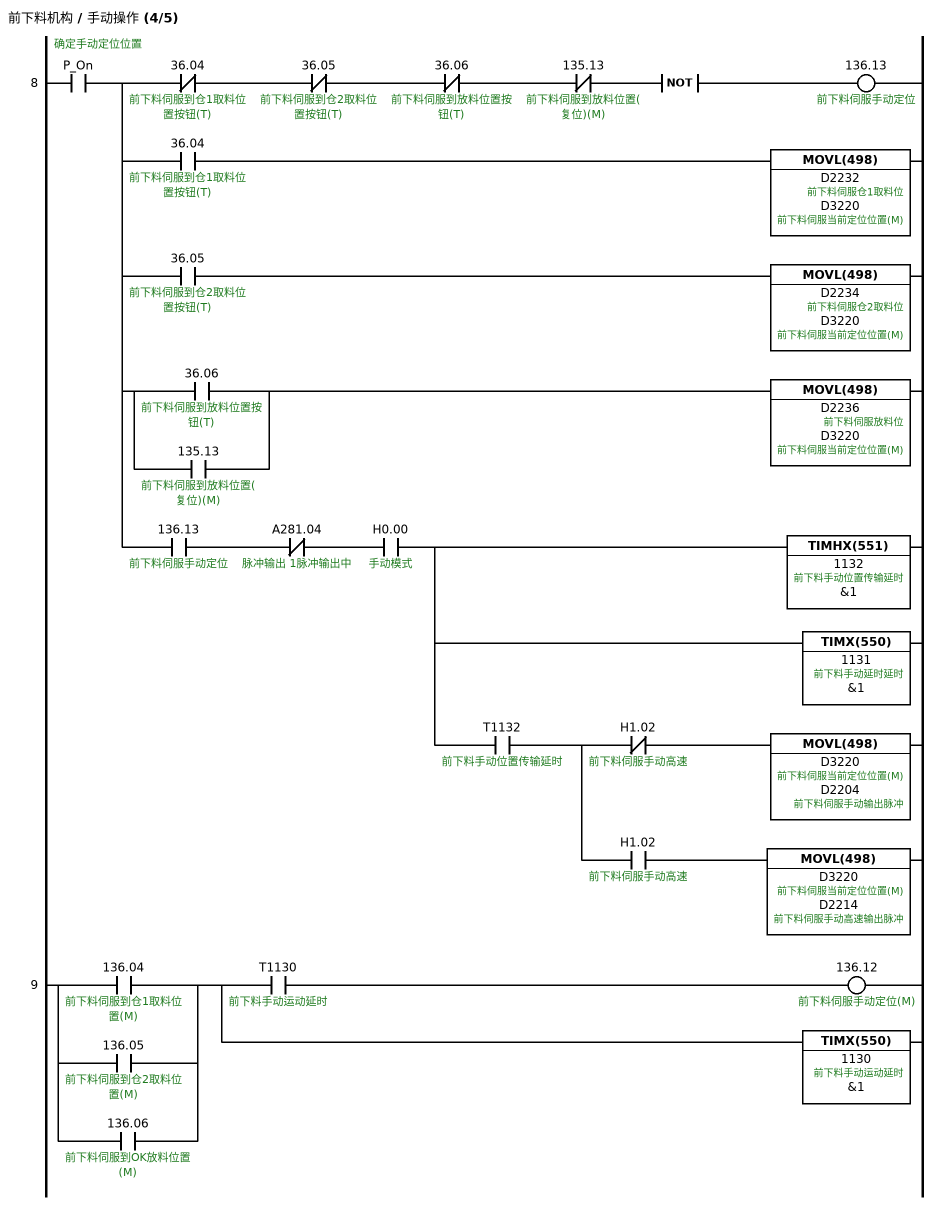
; [picture p168: 前下料机构 / 手动操作, rungs 8-9]
; rung 8: 确定手动定位位置
LD P_On
OUT TR0
ANDNOT 36.04  ; 前下料伺服到仓1取料位置按钮(T)
ANDNOT 36.05  ; 前下料伺服到仓2取料位置按钮(T)
ANDNOT 36.06  ; 前下料伺服到放料位置按钮(T)
ANDNOT 135.13  ; 前下料伺服到放料位置(复位)(M)
NOT(520)
OUT 136.13  ; 前下料伺服手动定位
LD TR0
AND 36.04  ; 前下料伺服到仓1取料位置按钮(T)
MOVL(498) D2232 D3220  ; 前下料伺服仓1取料位, 前下料伺服当前定位位置(M)
LD TR0
AND 36.05  ; 前下料伺服到仓2取料位置按钮(T)
MOVL(498) D2234 D3220  ; 前下料伺服仓2取料位, 前下料伺服当前定位位置(M)
LD TR0
LD 36.06  ; 前下料伺服到放料位置按钮(T)
OR 135.13  ; 前下料伺服到放料位置(复位)(M)
ANDLD
MOVL(498) D2236 D3220  ; 前下料伺服放料位, 前下料伺服当前定位位置(M)
LD TR0
AND 136.13  ; 前下料伺服手动定位
ANDNOT A281.04  ; 脉冲输出 1脉冲输出中
AND H0.00  ; 手动模式
TIMHX(551) 1132 &1  ; 前下料手动位置传输延时
TIMX(550) 1131 &1  ; 前下料手动延时延时
AND T1132  ; 前下料手动位置传输延时
OUT TR0
ANDNOT H1.02  ; 前下料伺服手动高速
MOVL(498) D3220 D2204  ; 前下料伺服当前定位位置(M), 前下料伺服手动输出脉冲
LD TR0
AND H1.02  ; 前下料伺服手动高速
MOVL(498) D3220 D2214  ; 前下料伺服当前定位位置(M), 前下料伺服手动高速输出脉冲
; rung 9
LD 136.04  ; 前下料伺服到仓1取料位置(M)
OR 136.05  ; 前下料伺服到仓2取料位置(M)
OR 136.06  ; 前下料伺服到OK放料位置(M)
OUT TR0
AND T1130  ; 前下料手动运动延时
OUT 136.12  ; 前下料伺服手动定位(M)
LD TR0
TIMX(550) 1130 &1  ; 前下料手动运动延时

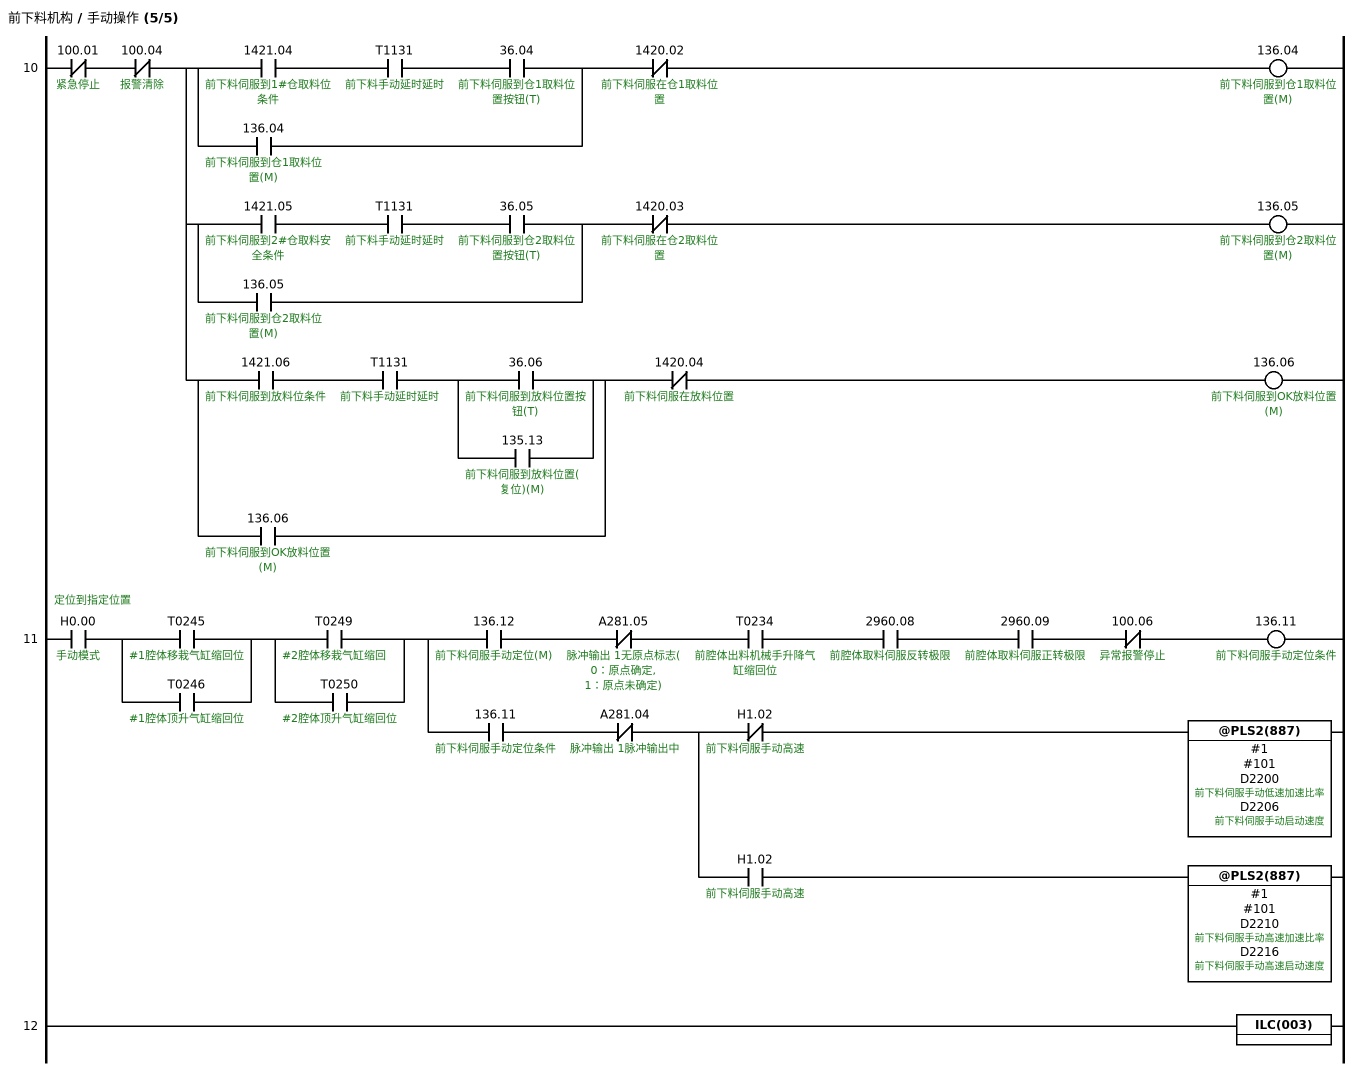
; rung 10
LDNOT 100.01  ; 紧急停止
ANDNOT 100.04  ; 报警清除
OUT TR0
LD 1421.04  ; 前下料伺服到1#仓取料位条件
AND T1131  ; 前下料手动延时延时
AND 36.04  ; 前下料伺服到仓1取料位置按钮(T)
OR 136.04  ; 前下料伺服到仓1取料位置(M)
ANDLD
ANDNOT 1420.02  ; 前下料伺服在仓1取料位置
OUT 136.04  ; 前下料伺服到仓1取料位置(M)
LD TR0
LD 1421.05  ; 前下料伺服到2#仓取料安全条件
AND T1131  ; 前下料手动延时延时
AND 36.05  ; 前下料伺服到仓2取料位置按钮(T)
OR 136.05  ; 前下料伺服到仓2取料位置(M)
ANDLD
ANDNOT 1420.03  ; 前下料伺服在仓2取料位置
OUT 136.05  ; 前下料伺服到仓2取料位置(M)
LD TR0
LD 1421.06  ; 前下料伺服到放料位条件
AND T1131  ; 前下料手动延时延时
LD 36.06  ; 前下料伺服到放料位置按钮(T)
OR 135.13  ; 前下料伺服到放料位置(复位)(M)
ANDLD
OR 136.06  ; 前下料伺服到OK放料位置(M)
ANDLD
ANDNOT 1420.04  ; 前下料伺服在放料位置
OUT 136.06  ; 前下料伺服到OK放料位置(M)
; rung 11: 定位到指定位置
LD H0.00  ; 手动模式
LD T0245  ; #1腔体移栽气缸缩回位
OR T0246  ; #1腔体顶升气缸缩回位
ANDLD
LD T0249  ; #2腔体移栽气缸缩回
OR T0250  ; #2腔体顶升气缸缩回位
ANDLD
OUT TR0
AND 136.12  ; 前下料伺服手动定位(M)
ANDNOT A281.05  ; 脉冲输出 1无原点标志(0：原点确定,1：原点未确定)
AND T0234  ; 前腔体出料机械手升降气缸缩回位
AND 2960.08  ; 前腔体取料伺服反转极限
AND 2960.09  ; 前腔体取料伺服正转极限
ANDNOT 100.06  ; 异常报警停止
OUT 136.11  ; 前下料伺服手动定位条件
LD TR0
AND 136.11  ; 前下料伺服手动定位条件
ANDNOT A281.04  ; 脉冲输出 1脉冲输出中
OUT TR0
ANDNOT H1.02  ; 前下料伺服手动高速
@PLS2(887) #1 #101 D2200 D2206  ; 前下料伺服手动低速加速比率, 前下料伺服手动启动速度
LD TR0
AND H1.02  ; 前下料伺服手动高速
@PLS2(887) #1 #101 D2210 D2216  ; 前下料伺服手动高速加速比率, 前下料伺服手动高速启动速度
; rung 12
ILC(003)

### Section 自动运行

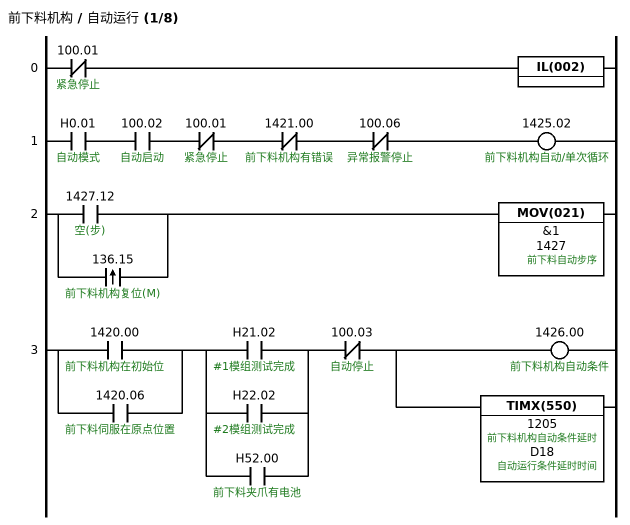
; rung 0
LDNOT 100.01  ; 紧急停止
IL(002)
; rung 1
LD H0.01  ; 自动模式
AND 100.02  ; 自动启动
ANDNOT 100.01  ; 紧急停止
ANDNOT 1421.00  ; 前下料机构有错误
ANDNOT 100.06  ; 异常报警停止
OUT 1425.02  ; 前下料机构自动/单次循环
; rung 2
LD 1427.12  ; 空(步)
@OR 136.15  ; 前下料机构复位(M)
MOV(021) &1 1427  ; 前下料自动步序
; rung 3
LD 1420.00  ; 前下料机构在初始位
OR 1420.06  ; 前下料伺服在原点位置
LD H21.02  ; #1模组测试完成
OR H22.02  ; #2模组测试完成
OR H52.00  ; 前下料夹爪有电池
ANDLD
ANDNOT 100.03  ; 自动停止
OUT 1426.00  ; 前下料机构自动条件
TIMX(550) 1205 D18  ; 自动运行条件延时时间, 前下料机构自动条件延时

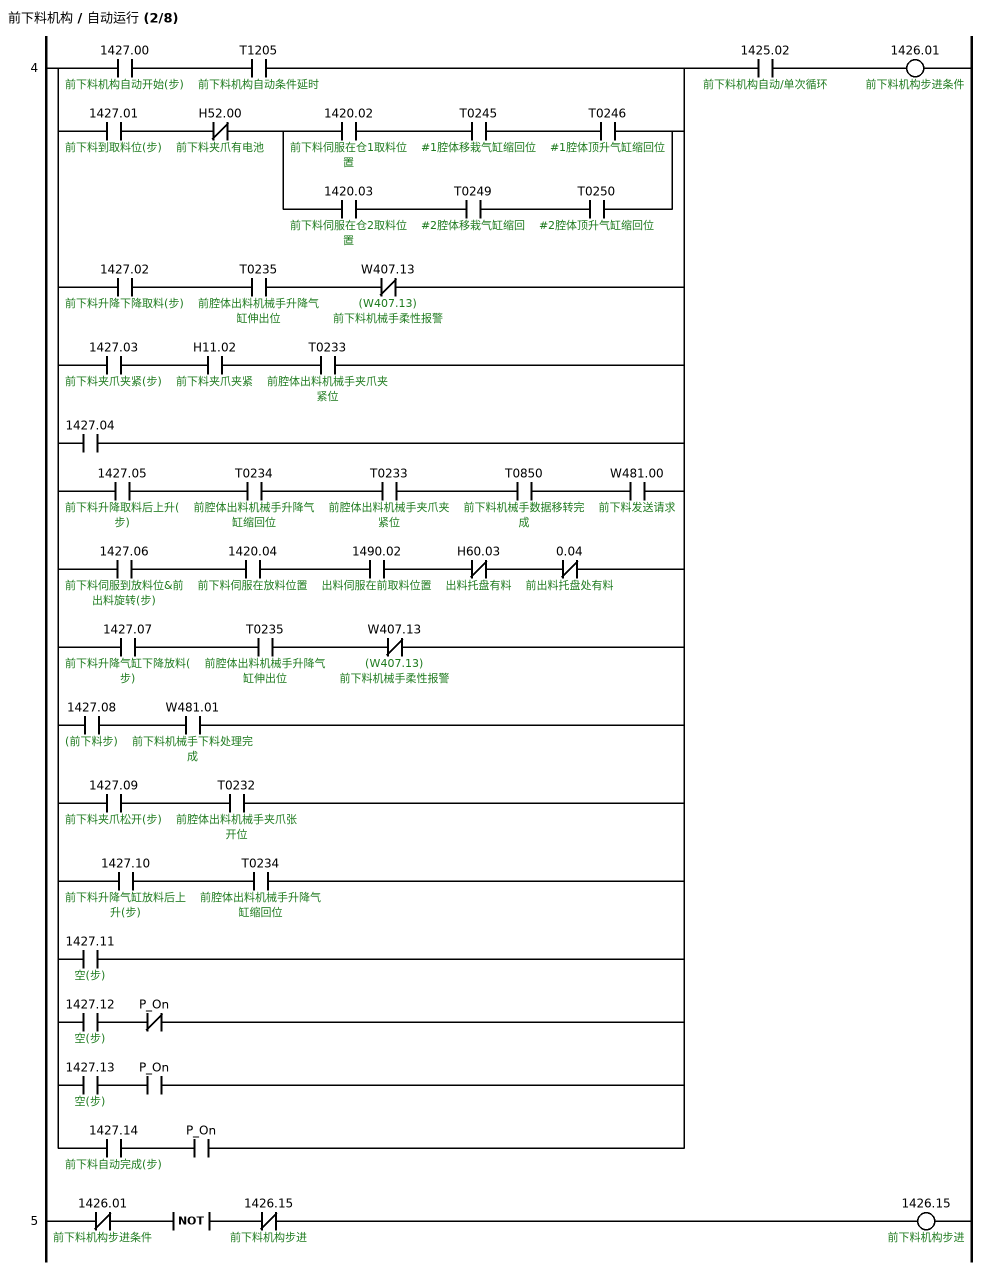
; rung 4
LD 1427.00  ; 前下料机构自动开始(步)
AND T1205  ; 前下料机构自动条件延时
LD 1427.01  ; 前下料到取料位(步)
ANDNOT H52.00  ; 前下料夹爪有电池
LD 1420.02  ; 前下料伺服在仓1取料位置
AND T0245  ; #1腔体移栽气缸缩回位
AND T0246  ; #1腔体顶升气缸缩回位
LD 1420.03  ; 前下料伺服在仓2取料位置
AND T0249  ; #2腔体移栽气缸缩回
AND T0250  ; #2腔体顶升气缸缩回位
ORLD
ANDLD
ORLD
LD 1427.02  ; 前下料升降下降取料(步)
AND T0235  ; 前腔体出料机械手升降气缸伸出位
ANDNOT W407.13  ; (W407.13) 前下料机械手柔性报警
ORLD
LD 1427.03  ; 前下料夹爪夹紧(步)
AND H11.02  ; 前下料夹爪夹紧
AND T0233  ; 前腔体出料机械手夹爪夹紧位
ORLD
OR 1427.04
LD 1427.05  ; 前下料升降取料后上升(步)
AND T0234  ; 前腔体出料机械手升降气缸缩回位
AND T0233  ; 前腔体出料机械手夹爪夹紧位
AND T0850  ; 前下料机械手数据移转完成
AND W481.00  ; 前下料发送请求
ORLD
LD 1427.06  ; 前下料伺服到放料位&前出料旋转(步)
AND 1420.04  ; 前下料伺服在放料位置
AND 1490.02  ; 出料伺服在前取料位置
ANDNOT H60.03  ; 出料托盘有料
ANDNOT 0.04  ; 前出料托盘处有料
ORLD
LD 1427.07  ; 前下料升降气缸下降放料(步)
AND T0235  ; 前腔体出料机械手升降气缸伸出位
ANDNOT W407.13  ; (W407.13) 前下料机械手柔性报警
ORLD
LD 1427.08  ; (前下料步)
AND W481.01  ; 前下料机械手下料处理完成
ORLD
LD 1427.09  ; 前下料夹爪松开(步)
AND T0232  ; 前腔体出料机械手夹爪张开位
ORLD
LD 1427.10  ; 前下料升降气缸放料后上升(步)
AND T0234  ; 前腔体出料机械手升降气缸缩回位
ORLD
OR 1427.11  ; 空(步)
LD 1427.12  ; 空(步)
ANDNOT P_On
ORLD
LD 1427.13  ; 空(步)
AND P_On
ORLD
LD 1427.14  ; 前下料自动完成(步)
AND P_On
ORLD
AND 1425.02  ; 前下料机构自动/单次循环
OUT 1426.01  ; 前下料机构步进条件
; rung 5
LDNOT 1426.01  ; 前下料机构步进条件
NOT(520)
ANDNOT 1426.15  ; 前下料机构步进
OUT 1426.15  ; 前下料机构步进

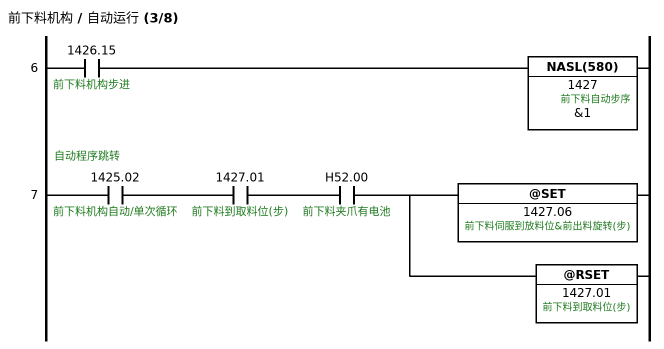
; rung 6
LD 1426.15  ; 前下料机构步进
NASL(580) 1427 &1  ; 前下料自动步序
; rung 7: 自动程序跳转
LD 1425.02  ; 前下料机构自动/单次循环
AND 1427.01  ; 前下料到取料位(步)
AND H52.00  ; 前下料夹爪有电池
@SET 1427.06  ; 前下料伺服到放料位&前出料旋转(步)
@RSET 1427.01  ; 前下料到取料位(步)

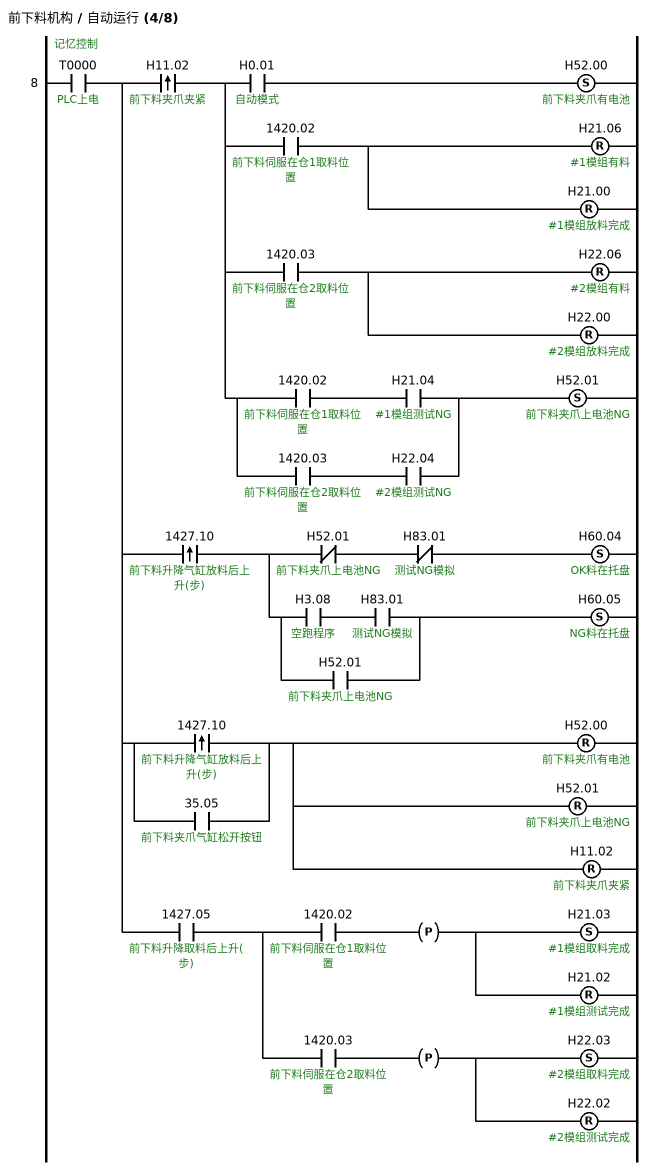
; rung 8: 记忆控制
LD T0000  ; PLC上电
OUT TR0
@AND H11.02  ; 前下料夹爪夹紧
OUT TR1
AND H0.01  ; 自动模式
SET H52.00  ; 前下料夹爪有电池
LD TR1
AND 1420.02  ; 前下料伺服在仓1取料位置
RSET H21.06  ; #1模组有料
RSET H21.00  ; #1模组放料完成
LD TR1
AND 1420.03  ; 前下料伺服在仓2取料位置
RSET H22.06  ; #2模组有料
RSET H22.00  ; #2模组放料完成
LD TR1
LD 1420.02  ; 前下料伺服在仓1取料位置
AND H21.04  ; #1模组测试NG
LD 1420.03  ; 前下料伺服在仓2取料位置
AND H22.04  ; #2模组测试NG
ORLD
ANDLD
SET H52.01  ; 前下料夹爪上电池NG
LD TR0
@AND 1427.10  ; 前下料升降气缸放料后上升(步)
OUT TR1
ANDNOT H52.01  ; 前下料夹爪上电池NG
ANDNOT H83.01  ; 测试NG模拟
SET H60.04  ; OK料在托盘
LD TR1
LD H3.08  ; 空跑程序
AND H83.01  ; 测试NG模拟
OR H52.01  ; 前下料夹爪上电池NG
ANDLD
SET H60.05  ; NG料在托盘
LD TR0
@LD 1427.10  ; 前下料升降气缸放料后上升(步)
OR 35.05  ; 前下料夹爪气缸松开按钮
ANDLD
RSET H52.00  ; 前下料夹爪有电池
RSET H52.01  ; 前下料夹爪上电池NG
RSET H11.02  ; 前下料夹爪夹紧
LD TR0
AND 1427.05  ; 前下料升降取料后上升(步)
OUT TR0
AND 1420.02  ; 前下料伺服在仓1取料位置
UP(521)
SET H21.03  ; #1模组取料完成
RSET H21.02  ; #1模组测试完成
LD TR0
AND 1420.03  ; 前下料伺服在仓2取料位置
UP(521)
SET H22.03  ; #2模组取料完成
RSET H22.02  ; #2模组测试完成

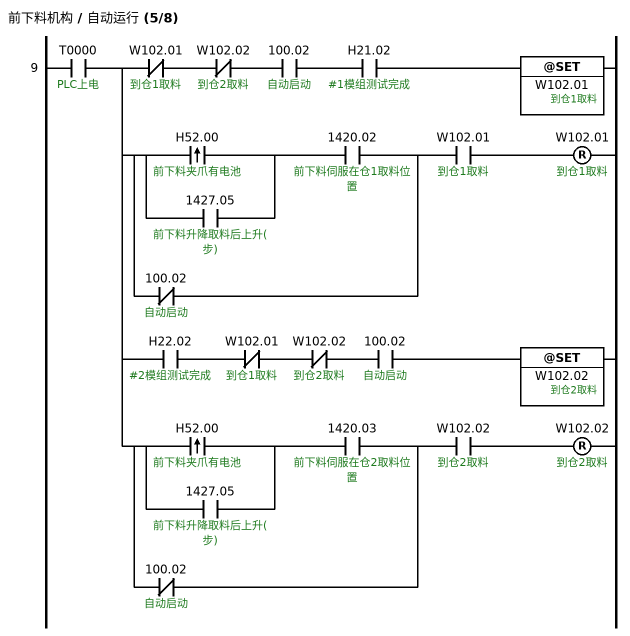
; rung 9
LD T0000  ; PLC上电
OUT TR0
ANDNOT W102.01  ; 到仓1取料
ANDNOT W102.02  ; 到仓2取料
AND 100.02  ; 自动启动
AND H21.02  ; #1模组测试完成
@SET W102.01  ; 到仓1取料
LD TR0
@LD H52.00  ; 前下料夹爪有电池
OR 1427.05  ; 前下料升降取料后上升(步)
AND 1420.02  ; 前下料伺服在仓1取料位置
ORNOT 100.02  ; 自动启动
ANDLD
AND W102.01  ; 到仓1取料
RSET W102.01  ; 到仓1取料
LD TR0
AND H22.02  ; #2模组测试完成
ANDNOT W102.01  ; 到仓1取料
ANDNOT W102.02  ; 到仓2取料
AND 100.02  ; 自动启动
@SET W102.02  ; 到仓2取料
LD TR0
@LD H52.00  ; 前下料夹爪有电池
OR 1427.05  ; 前下料升降取料后上升(步)
AND 1420.03  ; 前下料伺服在仓2取料位置
ORNOT 100.02  ; 自动启动
ANDLD
AND W102.02  ; 到仓2取料
RSET W102.02  ; 到仓2取料

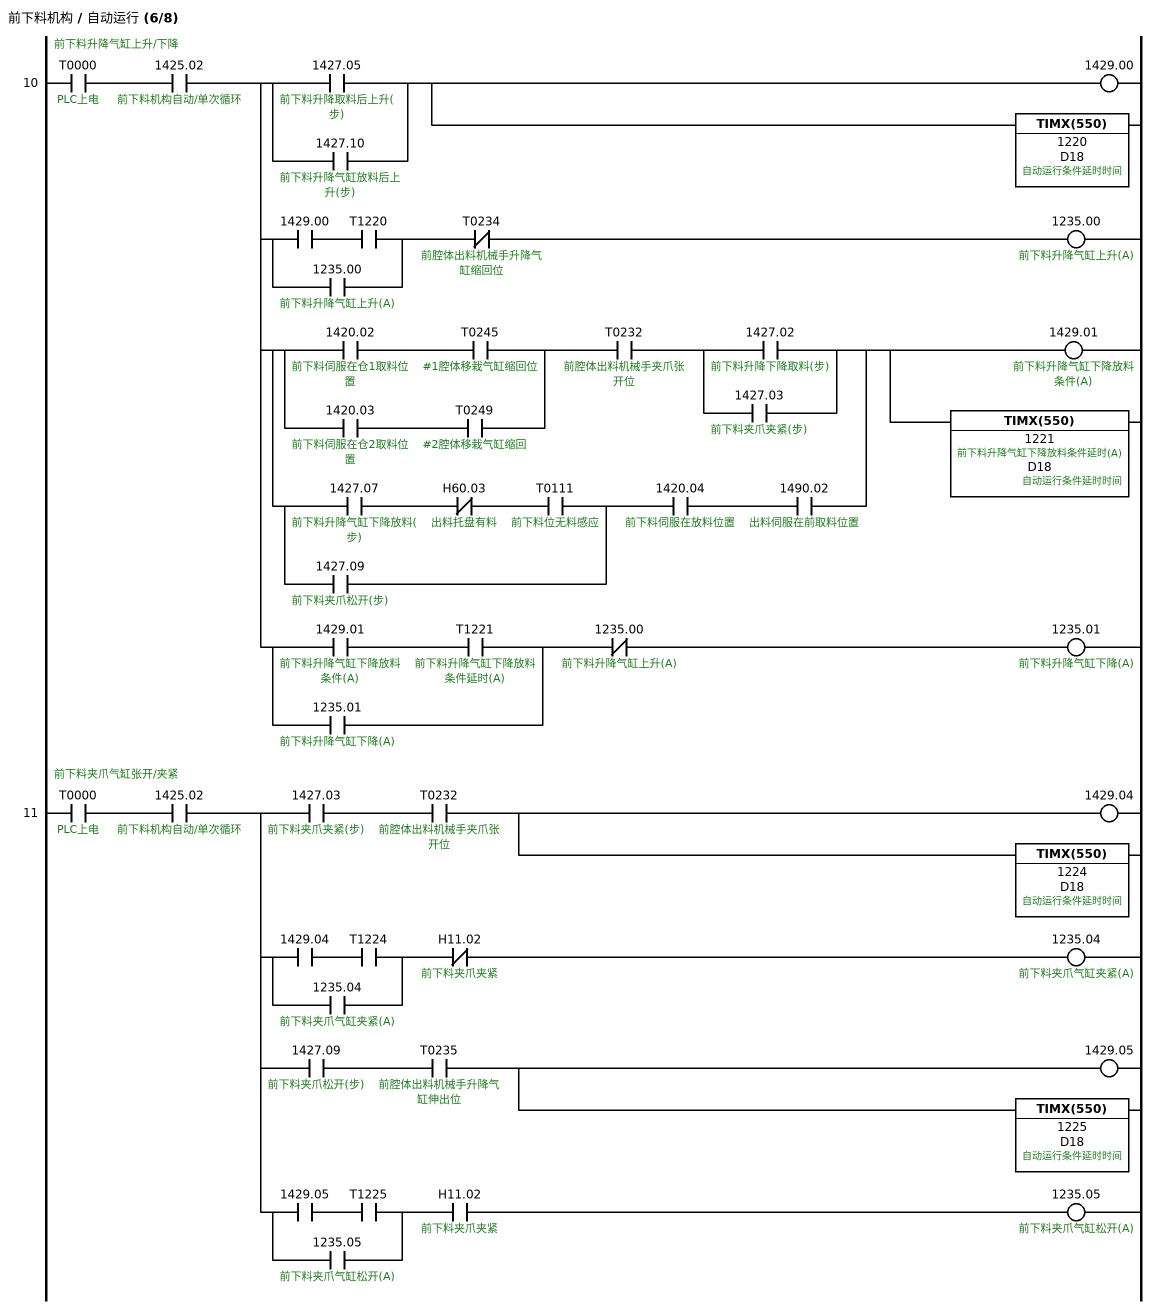
; rung 10: 前下料升降气缸上升/下降
LD T0000  ; PLC上电
AND 1425.02  ; 前下料机构自动/单次循环
OUT TR0
LD 1427.05  ; 前下料升降取料后上升(步)
OR 1427.10  ; 前下料升降气缸放料后上升(步)
ANDLD
OUT 1429.00
TIMX(550) 1220 D18  ; 自动运行条件延时时间
LD TR0
LD 1429.00
AND T1220
OR 1235.00  ; 前下料升降气缸上升(A)
ANDLD
ANDNOT T0234  ; 前腔体出料机械手升降气缸缩回位
OUT 1235.00  ; 前下料升降气缸上升(A)
LD TR0
LD 1420.02  ; 前下料伺服在仓1取料位置
AND T0245  ; #1腔体移栽气缸缩回位
LD 1420.03  ; 前下料伺服在仓2取料位置
AND T0249  ; #2腔体移栽气缸缩回
ORLD
AND T0232  ; 前腔体出料机械手夹爪张开位
LD 1427.02  ; 前下料升降下降取料(步)
OR 1427.03  ; 前下料夹爪夹紧(步)
ANDLD
LD 1427.07  ; 前下料升降气缸下降放料(步)
ANDNOT H60.03  ; 出料托盘有料
AND T0111  ; 前下料位无料感应
OR 1427.09  ; 前下料夹爪松开(步)
AND 1420.04  ; 前下料伺服在放料位置
AND 1490.02  ; 出料伺服在前取料位置
ORLD
ANDLD
OUT 1429.01  ; 前下料升降气缸下降放料条件(A)
TIMX(550) 1221 D18  ; 自动运行条件延时时间, 前下料升降气缸下降放料条件延时(A)
LD TR0
LD 1429.01  ; 前下料升降气缸下降放料条件(A)
AND T1221  ; 前下料升降气缸下降放料条件延时(A)
OR 1235.01  ; 前下料升降气缸下降(A)
ANDLD
ANDNOT 1235.00  ; 前下料升降气缸上升(A)
OUT 1235.01  ; 前下料升降气缸下降(A)
; rung 11: 前下料夹爪气缸张开/夹紧
LD T0000  ; PLC上电
AND 1425.02  ; 前下料机构自动/单次循环
OUT TR0
AND 1427.03  ; 前下料夹爪夹紧(步)
AND T0232  ; 前腔体出料机械手夹爪张开位
OUT 1429.04
TIMX(550) 1224 D18  ; 自动运行条件延时时间
LD TR0
LD 1429.04
AND T1224
OR 1235.04  ; 前下料夹爪气缸夹紧(A)
ANDLD
ANDNOT H11.02  ; 前下料夹爪夹紧
OUT 1235.04  ; 前下料夹爪气缸夹紧(A)
LD TR0
AND 1427.09  ; 前下料夹爪松开(步)
AND T0235  ; 前腔体出料机械手升降气缸伸出位
OUT 1429.05
TIMX(550) 1225 D18  ; 自动运行条件延时时间
LD TR0
LD 1429.05
AND T1225
OR 1235.05  ; 前下料夹爪气缸松开(A)
ANDLD
AND H11.02  ; 前下料夹爪夹紧
OUT 1235.05  ; 前下料夹爪气缸松开(A)

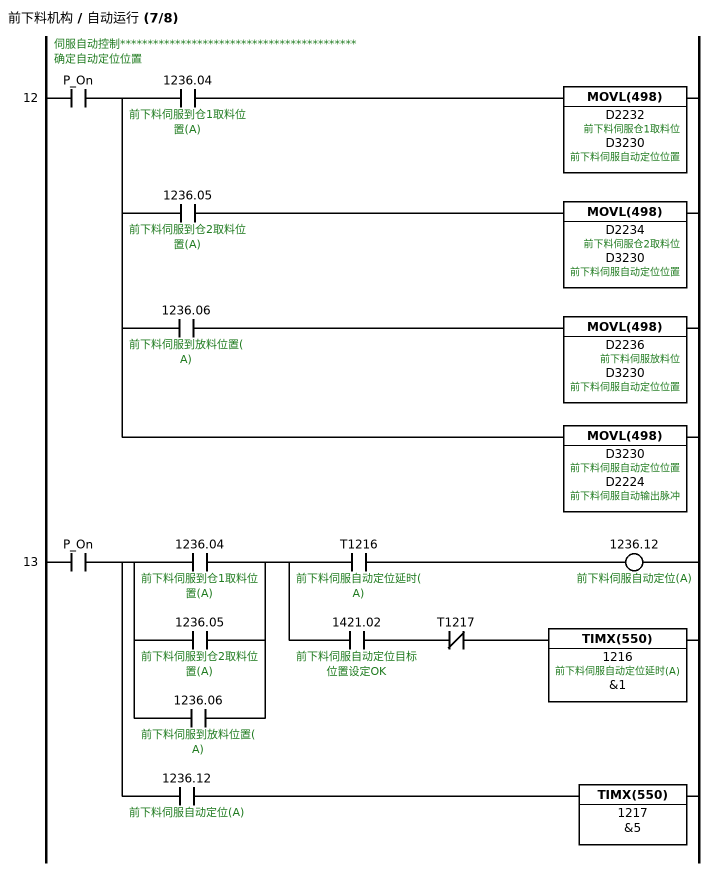
; rung 12: 伺服自动控制******************************************* / 确定自动定位位置
LD P_On
OUT TR0
AND 1236.04  ; 前下料伺服到仓1取料位置(A)
MOVL(498) D2232 D3230  ; 前下料伺服仓1取料位, 前下料伺服自动定位位置
LD TR0
AND 1236.05  ; 前下料伺服到仓2取料位置(A)
MOVL(498) D2234 D3230  ; 前下料伺服仓2取料位, 前下料伺服自动定位位置
LD TR0
AND 1236.06  ; 前下料伺服到放料位置(A)
MOVL(498) D2236 D3230  ; 前下料伺服放料位, 前下料伺服自动定位位置
LD TR0
MOVL(498) D3230 D2224  ; 前下料伺服自动定位位置, 前下料伺服自动输出脉冲
; rung 13
LD P_On
OUT TR0
LD 1236.04  ; 前下料伺服到仓1取料位置(A)
OR 1236.05  ; 前下料伺服到仓2取料位置(A)
OR 1236.06  ; 前下料伺服到放料位置(A)
ANDLD
OUT TR1
AND T1216  ; 前下料伺服自动定位延时(A)
OUT 1236.12  ; 前下料伺服自动定位(A)
LD TR1
AND 1421.02  ; 前下料伺服自动定位目标位置设定OK
ANDNOT T1217
TIMX(550) 1216 &1  ; 前下料伺服自动定位延时(A)
LD TR0
AND 1236.12  ; 前下料伺服自动定位(A)
TIMX(550) 1217 &5

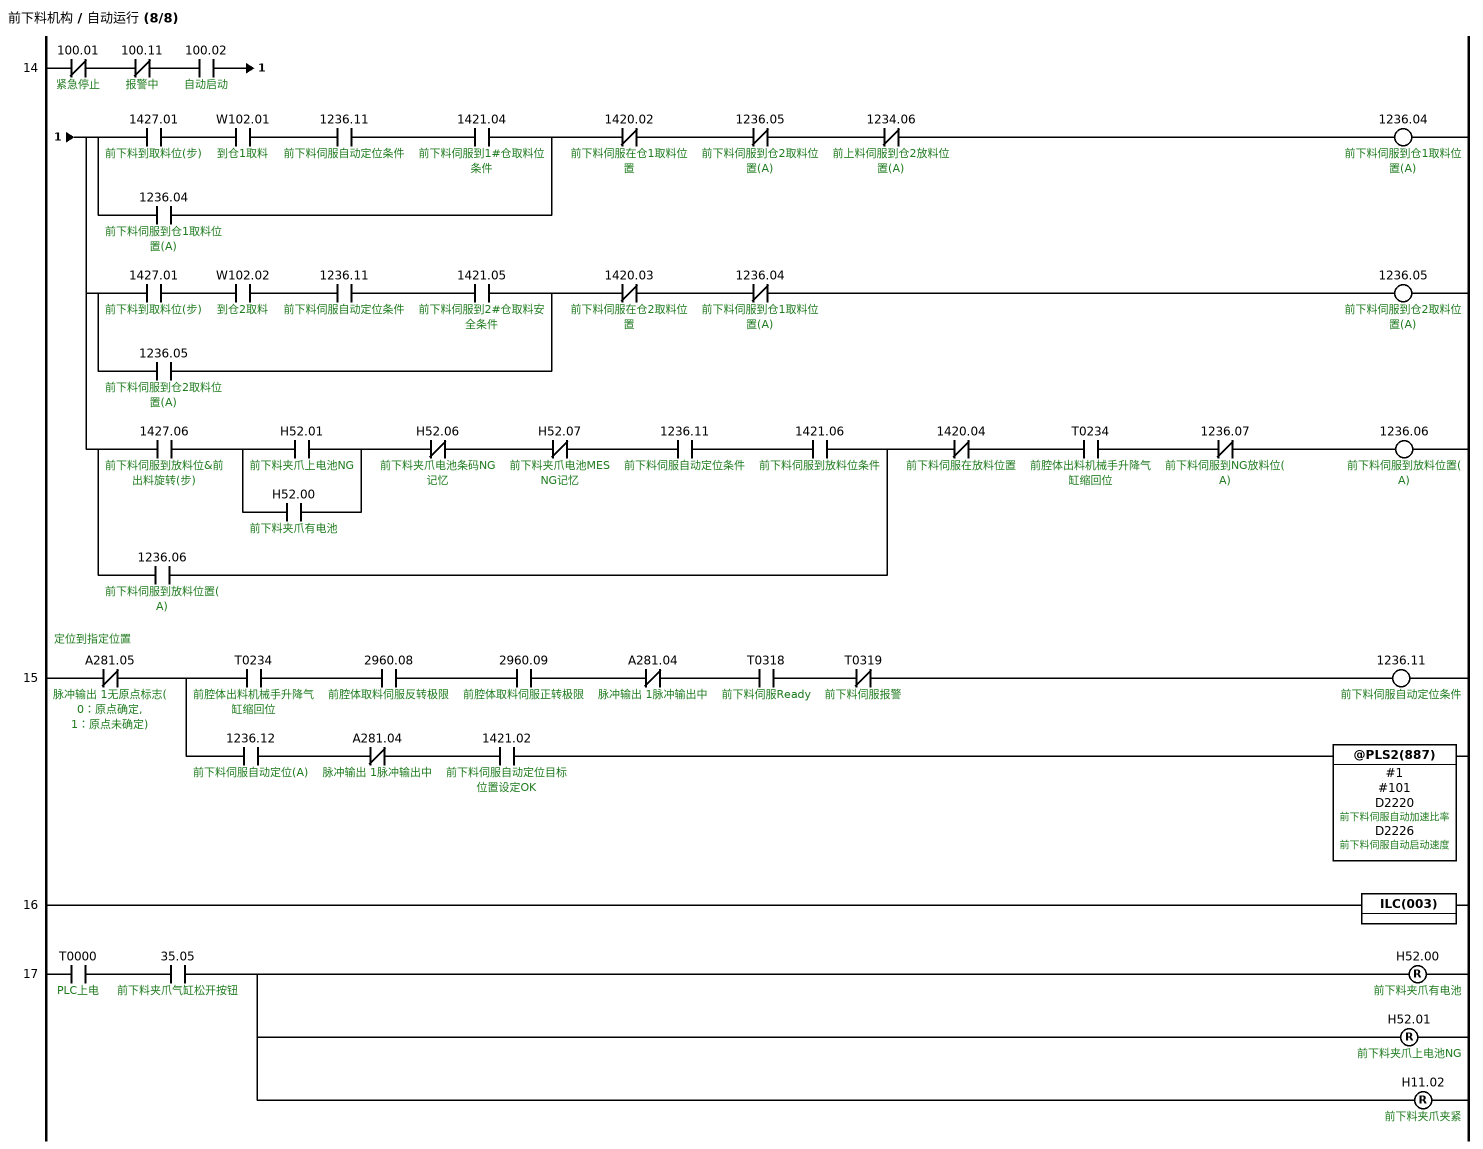
; rung 14
LDNOT 100.01  ; 紧急停止
ANDNOT 100.11  ; 报警中
AND 100.02  ; 自动启动
OUT TR0
LD 1427.01  ; 前下料到取料位(步)
AND W102.01  ; 到仓1取料
AND 1236.11  ; 前下料伺服自动定位条件
AND 1421.04  ; 前下料伺服到1#仓取料位条件
OR 1236.04  ; 前下料伺服到仓1取料位置(A)
ANDLD
ANDNOT 1420.02  ; 前下料伺服在仓1取料位置
ANDNOT 1236.05  ; 前下料伺服到仓2取料位置(A)
ANDNOT 1234.06  ; 前上料伺服到仓2放料位置(A)
OUT 1236.04  ; 前下料伺服到仓1取料位置(A)
LD TR0
LD 1427.01  ; 前下料到取料位(步)
AND W102.02  ; 到仓2取料
AND 1236.11  ; 前下料伺服自动定位条件
AND 1421.05  ; 前下料伺服到2#仓取料安全条件
OR 1236.05  ; 前下料伺服到仓2取料位置(A)
ANDLD
ANDNOT 1420.03  ; 前下料伺服在仓2取料位置
ANDNOT 1236.04  ; 前下料伺服到仓1取料位置(A)
OUT 1236.05  ; 前下料伺服到仓2取料位置(A)
LD TR0
LD 1427.06  ; 前下料伺服到放料位&前出料旋转(步)
LD H52.01  ; 前下料夹爪上电池NG
OR H52.00  ; 前下料夹爪有电池
ANDLD
ANDNOT H52.06  ; 前下料夹爪电池条码NG记忆
ANDNOT H52.07  ; 前下料夹爪电池MES NG记忆
AND 1236.11  ; 前下料伺服自动定位条件
AND 1421.06  ; 前下料伺服到放料位条件
OR 1236.06  ; 前下料伺服到放料位置(A)
ANDLD
ANDNOT 1420.04  ; 前下料伺服在放料位置
AND T0234  ; 前腔体出料机械手升降气缸缩回位
ANDNOT 1236.07  ; 前下料伺服到NG放料位(A)
OUT 1236.06  ; 前下料伺服到放料位置(A)
; rung 15: 定位到指定位置
LDNOT A281.05  ; 脉冲输出 1无原点标志(0：原点确定,1：原点未确定)
OUT TR0
AND T0234  ; 前腔体出料机械手升降气缸缩回位
AND 2960.08  ; 前腔体取料伺服反转极限
AND 2960.09  ; 前腔体取料伺服正转极限
ANDNOT A281.04  ; 脉冲输出 1脉冲输出中
AND T0318  ; 前下料伺服Ready
ANDNOT T0319  ; 前下料伺服报警
OUT 1236.11  ; 前下料伺服自动定位条件
LD TR0
AND 1236.12  ; 前下料伺服自动定位(A)
ANDNOT A281.04  ; 脉冲输出 1脉冲输出中
AND 1421.02  ; 前下料伺服自动定位目标位置设定OK
@PLS2(887) #1 #101 D2220 D2226  ; 前下料伺服自动加速比率, 前下料伺服自动启动速度
; rung 16
ILC(003)
; rung 17
LD T0000  ; PLC上电
AND 35.05  ; 前下料夹爪气缸松开按钮
RSET H52.00  ; 前下料夹爪有电池
RSET H52.01  ; 前下料夹爪上电池NG
RSET H11.02  ; 前下料夹爪夹紧

### Section 外部输出

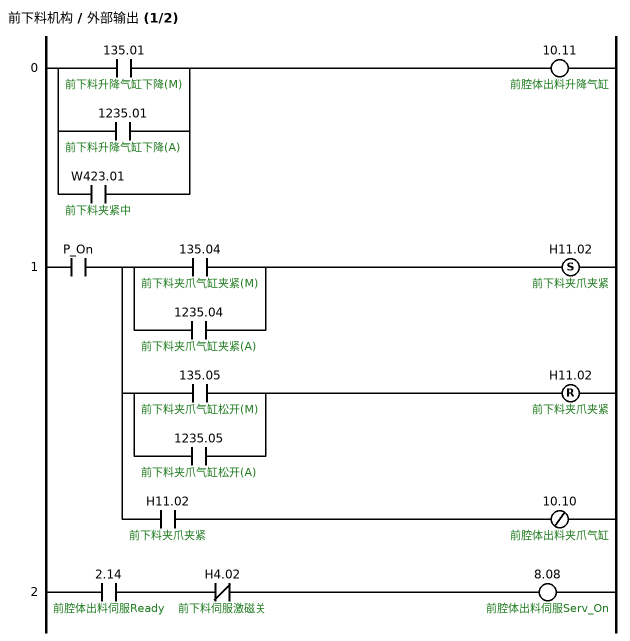
; rung 0
LD 135.01  ; 前下料升降气缸下降(M)
OR 1235.01  ; 前下料升降气缸下降(A)
OR W423.01  ; 前下料夹紧中
OUT 10.11  ; 前腔体出料升降气缸
; rung 1
LD P_On
OUT TR0
LD 135.04  ; 前下料夹爪气缸夹紧(M)
OR 1235.04  ; 前下料夹爪气缸夹紧(A)
ANDLD
SET H11.02  ; 前下料夹爪夹紧
LD TR0
LD 135.05  ; 前下料夹爪气缸松开(M)
OR 1235.05  ; 前下料夹爪气缸松开(A)
ANDLD
RSET H11.02  ; 前下料夹爪夹紧
LD TR0
AND H11.02  ; 前下料夹爪夹紧
OUTNOT 10.10  ; 前腔体出料夹爪气缸
; rung 2
LD 2.14  ; 前腔体出料伺服Ready
ANDNOT H4.02  ; 前下料伺服激磁关
OUT 8.08  ; 前腔体出料伺服Serv_On

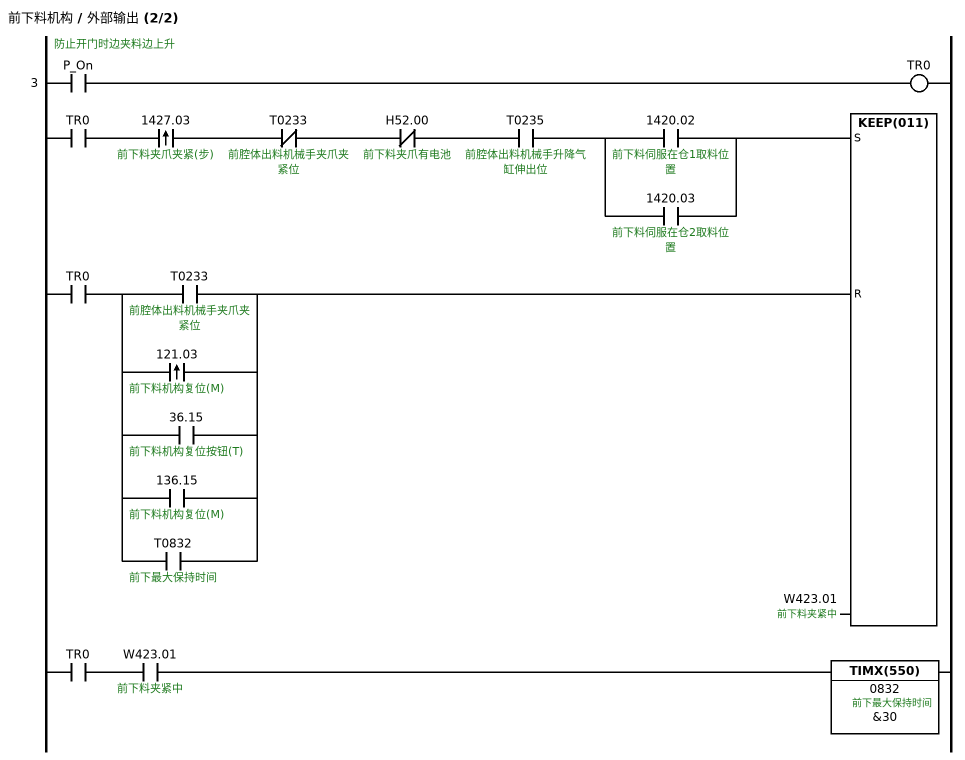
; rung 3: 防止开门时边夹料边上升
LD P_On
OUT TR0
@AND 1427.03  ; 前下料夹爪夹紧(步)
ANDNOT T0233  ; 前腔体出料机械手夹爪夹紧位
ANDNOT H52.00  ; 前下料夹爪有电池
AND T0235  ; 前腔体出料机械手升降气缸伸出位
LD 1420.02  ; 前下料伺服在仓1取料位置
OR 1420.03  ; 前下料伺服在仓2取料位置
ANDLD
LD TR0
LD T0233  ; 前腔体出料机械手夹爪夹紧位
@OR 121.03  ; 前下料机构复位(M)
OR 36.15  ; 前下料机构复位按钮(T)
OR 136.15  ; 前下料机构复位(M)
OR T0832  ; 前下最大保持时间
ANDLD
KEEP(011) W423.01  ; 前下料夹紧中
LD TR0
AND W423.01  ; 前下料夹紧中
TIMX(550) 0832 &30  ; 前下最大保持时间

### Section 进出机构外部输出

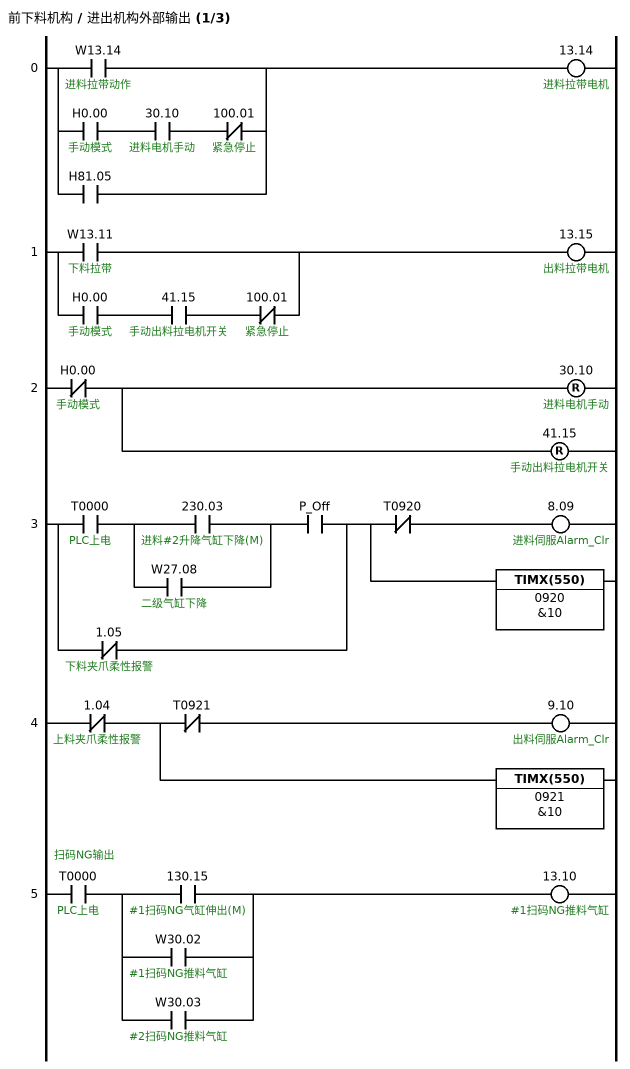
; rung 0
LD W13.14  ; 进料拉带动作
LD H0.00  ; 手动模式
AND 30.10  ; 进料电机手动
ANDNOT 100.01  ; 紧急停止
ORLD
OR H81.05
OUT 13.14  ; 进料拉带电机
; rung 1
LD W13.11  ; 下料拉带
LD H0.00  ; 手动模式
AND 41.15  ; 手动出料拉电机开关
ANDNOT 100.01  ; 紧急停止
ORLD
OUT 13.15  ; 出料拉带电机
; rung 2
LDNOT H0.00  ; 手动模式
RSET 30.10  ; 进料电机手动
RSET 41.15  ; 手动出料拉电机开关
; rung 3
LD T0000  ; PLC上电
LD 230.03  ; 进料#2升降气缸下降(M)
OR W27.08  ; 二级气缸下降
ANDLD
AND P_Off
ORNOT 1.05  ; 下料夹爪柔性报警
OUT TR0
ANDNOT T0920
OUT 8.09  ; 进料伺服Alarm_Clr
LD TR0
TIMX(550) 0920 &10
; rung 4
LDNOT 1.04  ; 上料夹爪柔性报警
OUT TR0
ANDNOT T0921
OUT 9.10  ; 出料伺服Alarm_Clr
LD TR0
TIMX(550) 0921 &10
; rung 5: 扫码NG输出
LD T0000  ; PLC上电
LD 130.15  ; #1扫码NG气缸伸出(M)
OR W30.02  ; #1扫码NG推料气缸
OR W30.03  ; #2扫码NG推料气缸
ANDLD
OUT 13.10  ; #1扫码NG推料气缸

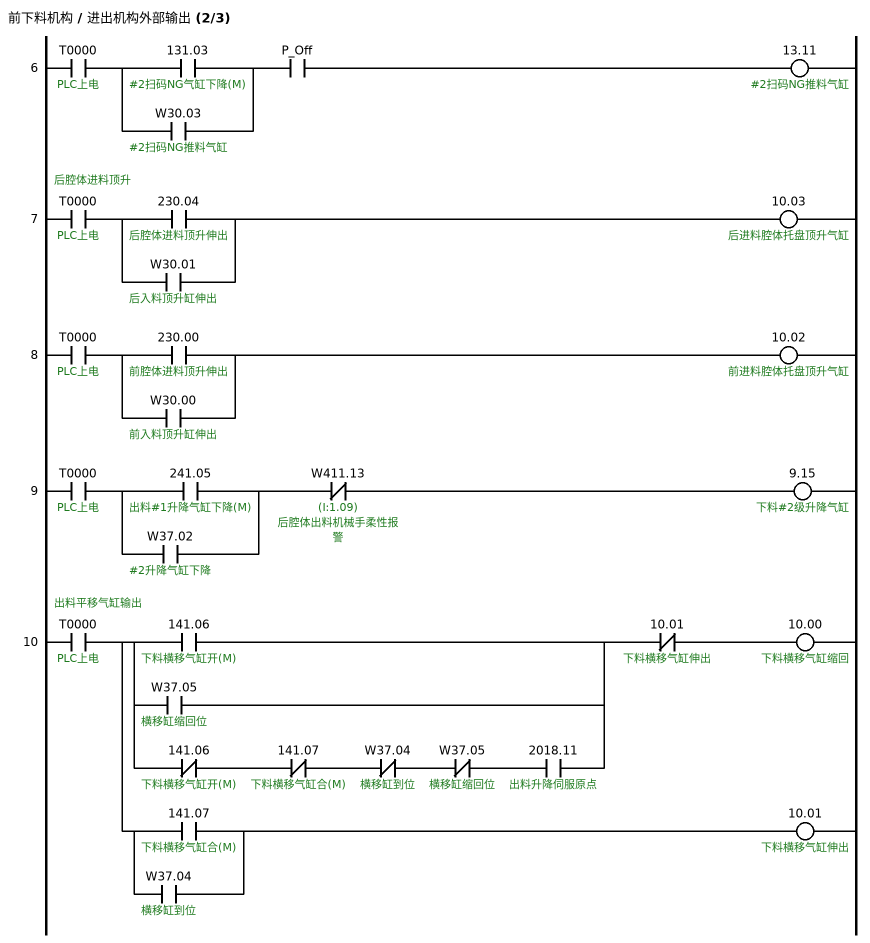
; rung 6
LD T0000  ; PLC上电
LD 131.03  ; #2扫码NG气缸下降(M)
OR W30.03  ; #2扫码NG推料气缸
ANDLD
AND P_Off
OUT 13.11  ; #2扫码NG推料气缸
; rung 7: 后腔体进料顶升
LD T0000  ; PLC上电
LD 230.04  ; 后腔体进料顶升伸出
OR W30.01  ; 后入料顶升缸伸出
ANDLD
OUT 10.03  ; 后进料腔体托盘顶升气缸
; rung 8
LD T0000  ; PLC上电
LD 230.00  ; 前腔体进料顶升伸出
OR W30.00  ; 前入料顶升缸伸出
ANDLD
OUT 10.02  ; 前进料腔体托盘顶升气缸
; rung 9
LD T0000  ; PLC上电
LD 241.05  ; 出料#1升降气缸下降(M)
OR W37.02  ; #2升降气缸下降
ANDLD
ANDNOT W411.13  ; (I:1.09) 后腔体出料机械手柔性报警
OUT 9.15  ; 下料#2级升降气缸
; rung 10: 出料平移气缸输出
LD T0000  ; PLC上电
OUT TR0
LD 141.06  ; 下料横移气缸开(M)
OR W37.05  ; 横移缸缩回位
LDNOT 141.06  ; 下料横移气缸开(M)
ANDNOT 141.07  ; 下料横移气缸合(M)
ANDNOT W37.04  ; 横移缸到位
ANDNOT W37.05  ; 横移缸缩回位
AND 2018.11  ; 出料升降伺服原点
ORLD
ANDLD
ANDNOT 10.01  ; 下料横移气缸伸出
OUT 10.00  ; 下料横移气缸缩回
LD TR0
LD 141.07  ; 下料横移气缸合(M)
OR W37.04  ; 横移缸到位
ANDLD
OUT 10.01  ; 下料横移气缸伸出

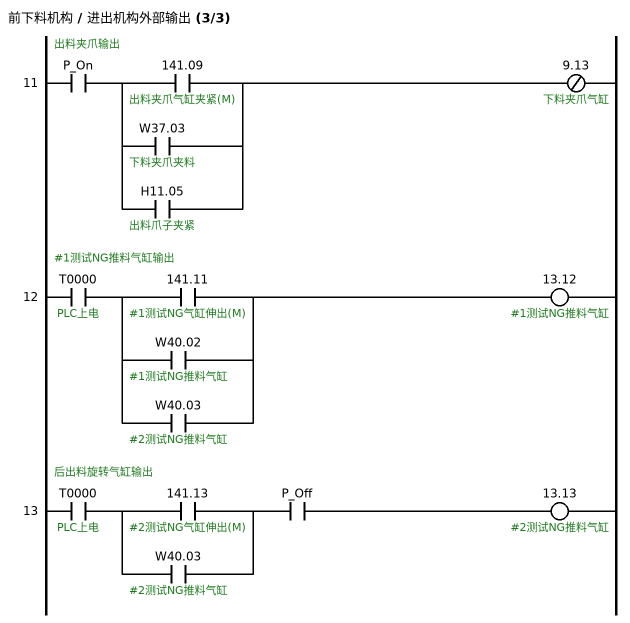
; rung 11: 出料夹爪输出
LD P_On
LD 141.09  ; 出料夹爪气缸夹紧(M)
OR W37.03  ; 下料夹爪夹料
OR H11.05  ; 出料爪子夹紧
ANDLD
OUTNOT 9.13  ; 下料夹爪气缸
; rung 12: #1测试NG推料气缸输出
LD T0000  ; PLC上电
LD 141.11  ; #1测试NG气缸伸出(M)
OR W40.02  ; #1测试NG推料气缸
OR W40.03  ; #2测试NG推料气缸
ANDLD
OUT 13.12  ; #1测试NG推料气缸
; rung 13: 后出料旋转气缸输出
LD T0000  ; PLC上电
LD 141.13  ; #2测试NG气缸伸出(M)
OR W40.03  ; #2测试NG推料气缸
ANDLD
AND P_Off
OUT 13.13  ; #2测试NG推料气缸

### Section 指示灯
; rung 0: ************************************************** / 气缸动作及位置指示灯

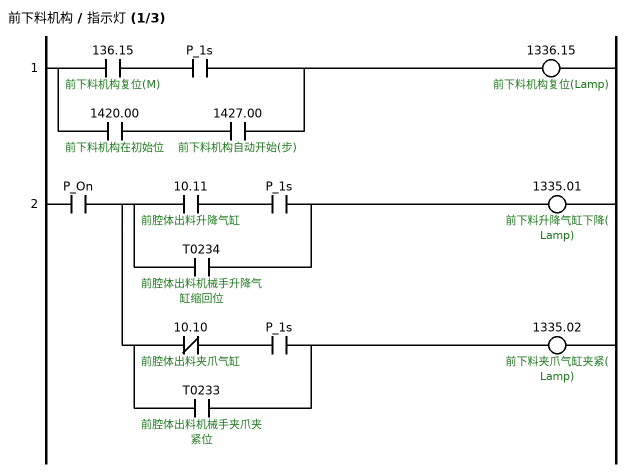
; rung 1
LD 136.15  ; 前下料机构复位(M)
AND P_1s
LD 1420.00  ; 前下料机构在初始位
AND 1427.00  ; 前下料机构自动开始(步)
ORLD
OUT 1336.15  ; 前下料机构复位(Lamp)
; rung 2
LD P_On
OUT TR0
LD 10.11  ; 前腔体出料升降气缸
AND P_1s
OR T0234  ; 前腔体出料机械手升降气缸缩回位
ANDLD
OUT 1335.01  ; 前下料升降气缸下降(Lamp)
LD TR0
LDNOT 10.10  ; 前腔体出料夹爪气缸
AND P_1s
OR T0233  ; 前腔体出料机械手夹爪夹紧位
ANDLD
OUT 1335.02  ; 前下料夹爪气缸夹紧(Lamp)

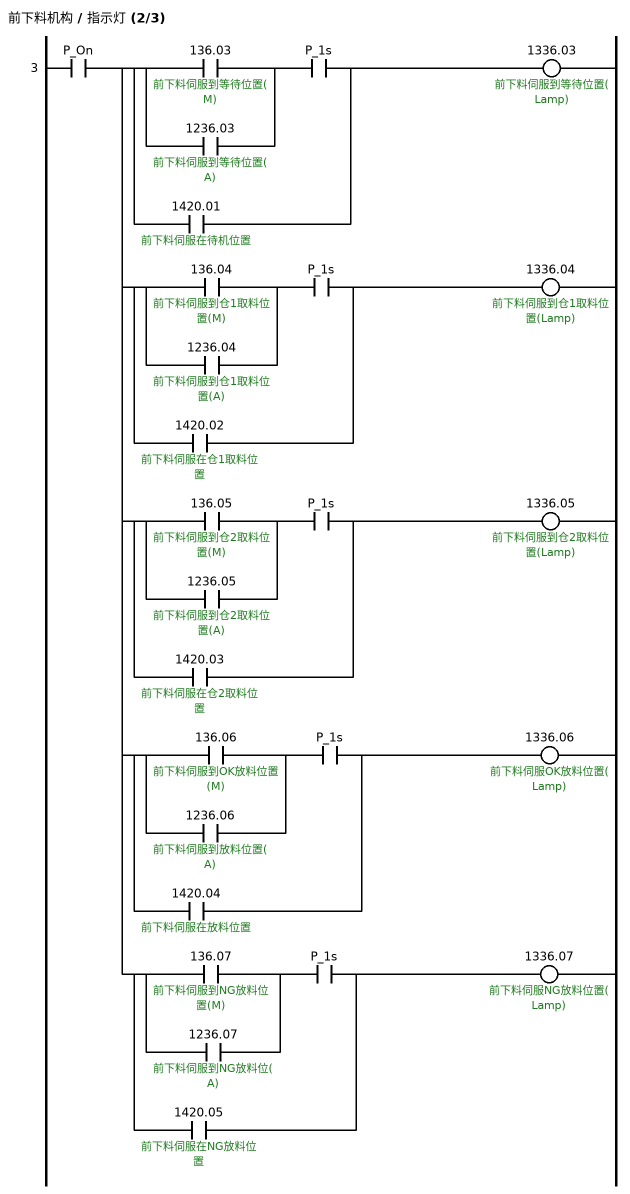
; rung 3
LD P_On
OUT TR0
LD 136.03  ; 前下料伺服到等待位置(M)
OR 1236.03  ; 前下料伺服到等待位置(A)
AND P_1s
OR 1420.01  ; 前下料伺服在待机位置
ANDLD
OUT 1336.03  ; 前下料伺服到等待位置(Lamp)
LD TR0
LD 136.04  ; 前下料伺服到仓1取料位置(M)
OR 1236.04  ; 前下料伺服到仓1取料位置(A)
AND P_1s
OR 1420.02  ; 前下料伺服在仓1取料位置
ANDLD
OUT 1336.04  ; 前下料伺服到仓1取料位置(Lamp)
LD TR0
LD 136.05  ; 前下料伺服到仓2取料位置(M)
OR 1236.05  ; 前下料伺服到仓2取料位置(A)
AND P_1s
OR 1420.03  ; 前下料伺服在仓2取料位置
ANDLD
OUT 1336.05  ; 前下料伺服到仓2取料位置(Lamp)
LD TR0
LD 136.06  ; 前下料伺服到OK放料位置(M)
OR 1236.06  ; 前下料伺服到放料位置(A)
AND P_1s
OR 1420.04  ; 前下料伺服在放料位置
ANDLD
OUT 1336.06  ; 前下料伺服OK放料位置(Lamp)
LD TR0
LD 136.07  ; 前下料伺服到NG放料位置(M)
OR 1236.07  ; 前下料伺服到NG放料位(A)
AND P_1s
OR 1420.05  ; 前下料伺服在NG放料位置
ANDLD
OUT 1336.07  ; 前下料伺服NG放料位置(Lamp)

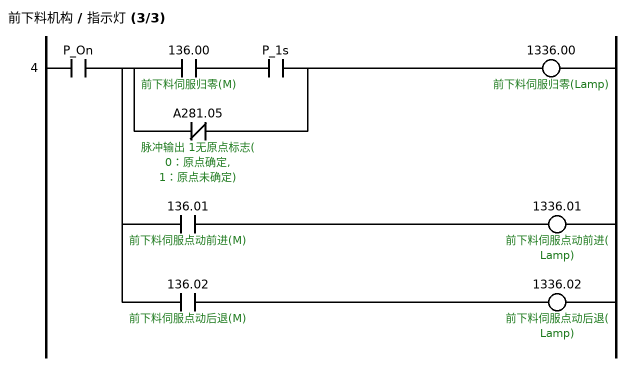
; rung 4
LD P_On
OUT TR0
LD 136.00  ; 前下料伺服归零(M)
AND P_1s
ORNOT A281.05  ; 脉冲输出 1无原点标志(0：原点确定,1：原点未确定)
ANDLD
OUT 1336.00  ; 前下料伺服归零(Lamp)
LD TR0
AND 136.01  ; 前下料伺服点动前进(M)
OUT 1336.01  ; 前下料伺服点动前进(Lamp)
LD TR0
AND 136.02  ; 前下料伺服点动后退(M)
OUT 1336.02  ; 前下料伺服点动后退(Lamp)

### Section END
; rung 0
END(001)

## Program 后上料机构 (cyclic task 4)

### Section Main

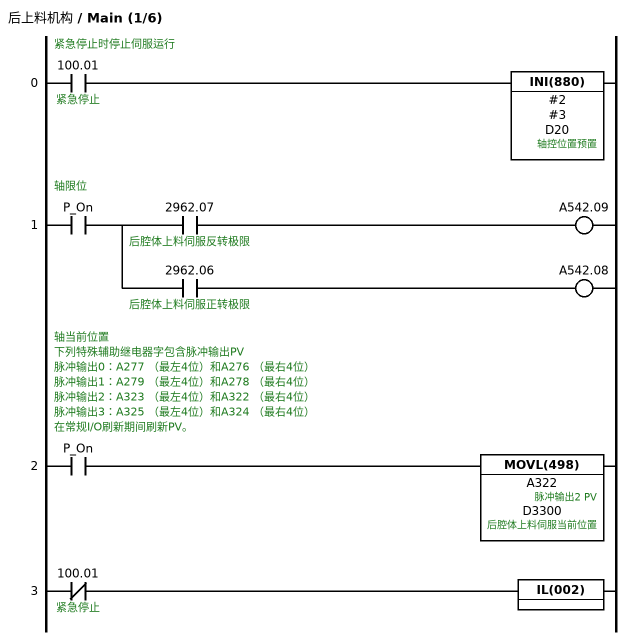
; rung 0: 紧急停止时停止伺服运行
LD 100.01  ; 紧急停止
INI(880) #2 #3 D20  ; 轴控位置预置
; rung 1: 轴限位
LD P_On
OUT TR0
AND 2962.07  ; 后腔体上料伺服反转极限
OUT A542.09
LD TR0
AND 2962.06  ; 后腔体上料伺服正转极限
OUT A542.08
; rung 2: 轴当前位置 / 下列特殊辅助继电器字包含脉冲输出PV / 脉冲输出0：A277 （最左4位）和A276 （最右4位） / 脉冲输出1：A279 （最左4位）和A278 （最右4位） / 脉冲输出2：A323 （最左4位）和A322 （最右4位） / 脉冲输出3：A325 （最左4位）和A324 （最右4位） / 在常规I/O刷新期间刷新PV。
LD P_On
MOVL(498) A322 D3300  ; 脉冲输出2 PV, 后腔体上料伺服当前位置
; rung 3
LDNOT 100.01  ; 紧急停止
IL(002)

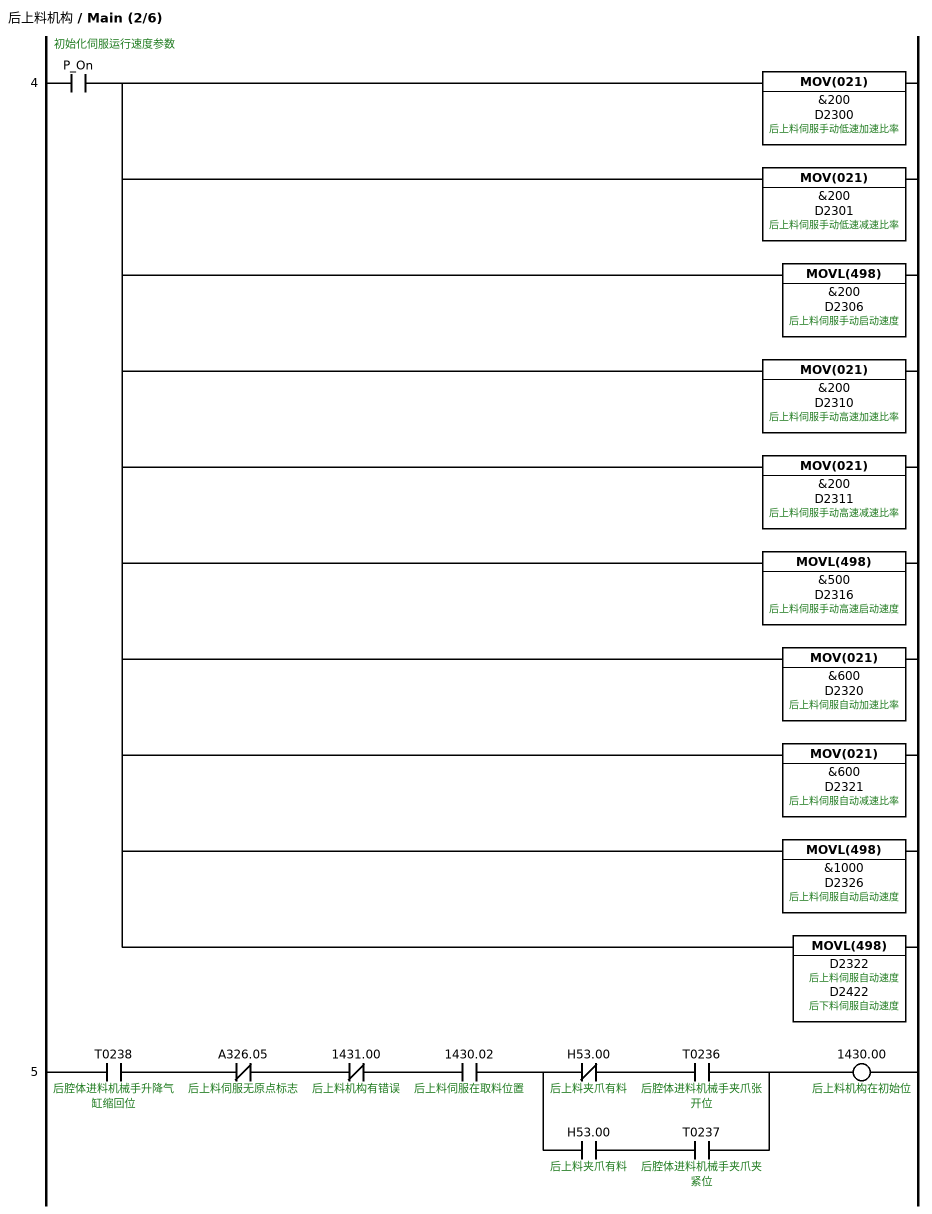
; rung 4: 初始化伺服运行速度参数
LD P_On
MOV(021) &200 D2300  ; 后上料伺服手动低速加速比率
MOV(021) &200 D2301  ; 后上料伺服手动低速减速比率
MOVL(498) &200 D2306  ; 后上料伺服手动启动速度
MOV(021) &200 D2310  ; 后上料伺服手动高速加速比率
MOV(021) &200 D2311  ; 后上料伺服手动高速减速比率
MOVL(498) &500 D2316  ; 后上料伺服手动高速启动速度
MOV(021) &600 D2320  ; 后上料伺服自动加速比率
MOV(021) &600 D2321  ; 后上料伺服自动减速比率
MOVL(498) &1000 D2326  ; 后上料伺服自动启动速度
MOVL(498) D2322 D2422  ; 后上料伺服自动速度, 后下料伺服自动速度
; rung 5
LD T0238  ; 后腔体进料机械手升降气缸缩回位
ANDNOT A326.05  ; 后上料伺服无原点标志
ANDNOT 1431.00  ; 后上料机构有错误
AND 1430.02  ; 后上料伺服在取料位置
LDNOT H53.00  ; 后上料夹爪有料
AND T0236  ; 后腔体进料机械手夹爪张开位
LD H53.00  ; 后上料夹爪有料
AND T0237  ; 后腔体进料机械手夹爪夹紧位
ORLD
ANDLD
OUT 1430.00  ; 后上料机构在初始位

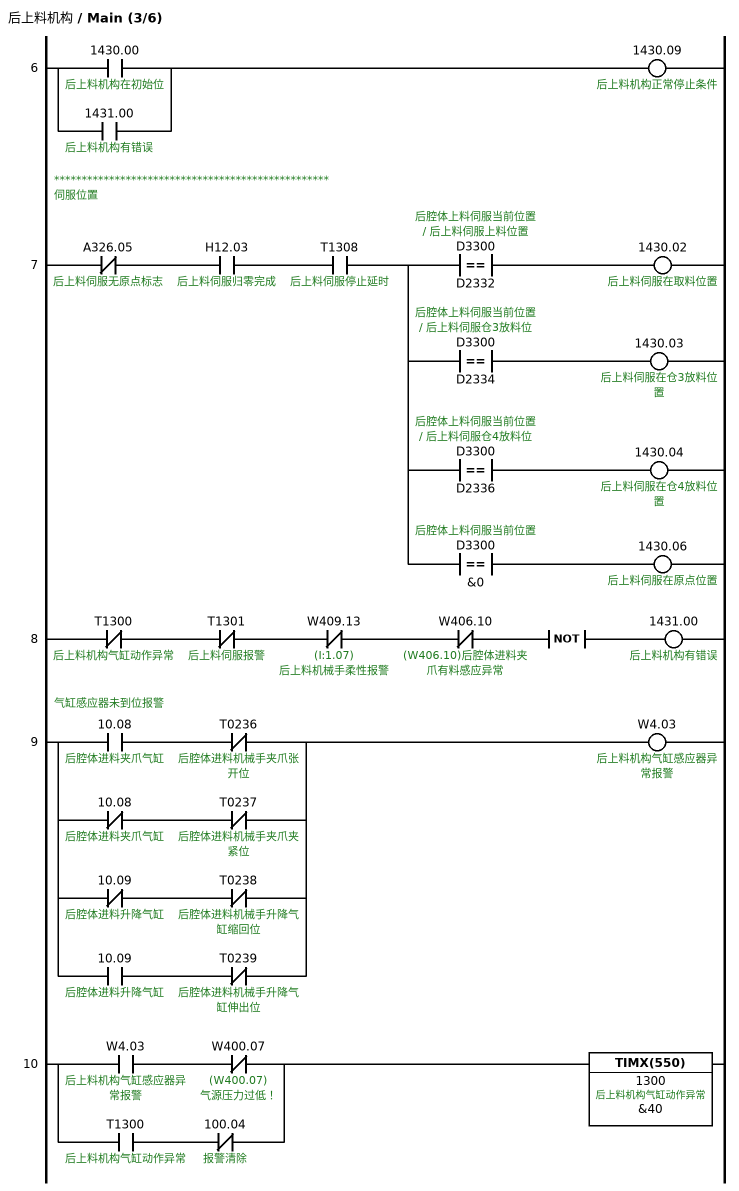
; rung 6
LD 1430.00  ; 后上料机构在初始位
OR 1431.00  ; 后上料机构有错误
OUT 1430.09  ; 后上料机构正常停止条件
; rung 7: ************************************************** / 伺服位置
LDNOT A326.05  ; 后上料伺服无原点标志
AND H12.03  ; 后上料伺服归零完成
AND T1308  ; 后上料伺服停止延时
OUT TR0
AND=SL(303) D3300 D2332  ; 后腔体上料伺服当前位置, 后上料伺服上料位置
OUT 1430.02  ; 后上料伺服在取料位置
LD TR0
AND=SL(303) D3300 D2334  ; 后腔体上料伺服当前位置, 后上料伺服仓3放料位
OUT 1430.03  ; 后上料伺服在仓3放料位置
LD TR0
AND=SL(303) D3300 D2336  ; 后腔体上料伺服当前位置, 后上料伺服仓4放料位
OUT 1430.04  ; 后上料伺服在仓4放料位置
LD TR0
AND=SL(303) D3300 &0  ; 后腔体上料伺服当前位置
OUT 1430.06  ; 后上料伺服在原点位置
; rung 8
LDNOT T1300  ; 后上料机构气缸动作异常
ANDNOT T1301  ; 后上料伺服报警
ANDNOT W409.13  ; (I:1.07) 后上料机械手柔性报警
ANDNOT W406.10  ; (W406.10)后腔体进料夹爪有料感应异常
NOT(520)
OUT 1431.00  ; 后上料机构有错误
; rung 9: 气缸感应器未到位报警
LD 10.08  ; 后腔体进料夹爪气缸
ANDNOT T0236  ; 后腔体进料机械手夹爪张开位
LDNOT 10.08  ; 后腔体进料夹爪气缸
ANDNOT T0237  ; 后腔体进料机械手夹爪夹紧位
ORLD
LDNOT 10.09  ; 后腔体进料升降气缸
ANDNOT T0238  ; 后腔体进料机械手升降气缸缩回位
ORLD
LD 10.09  ; 后腔体进料升降气缸
ANDNOT T0239  ; 后腔体进料机械手升降气缸伸出位
ORLD
OUT W4.03  ; 后上料机构气缸感应器异常报警
; rung 10
LD W4.03  ; 后上料机构气缸感应器异常报警
ANDNOT W400.07  ; (W400.07) 气源压力过低！
LD T1300  ; 后上料机构气缸动作异常
ANDNOT 100.04  ; 报警清除
ORLD
TIMX(550) 1300 &40  ; 后上料机构气缸动作异常

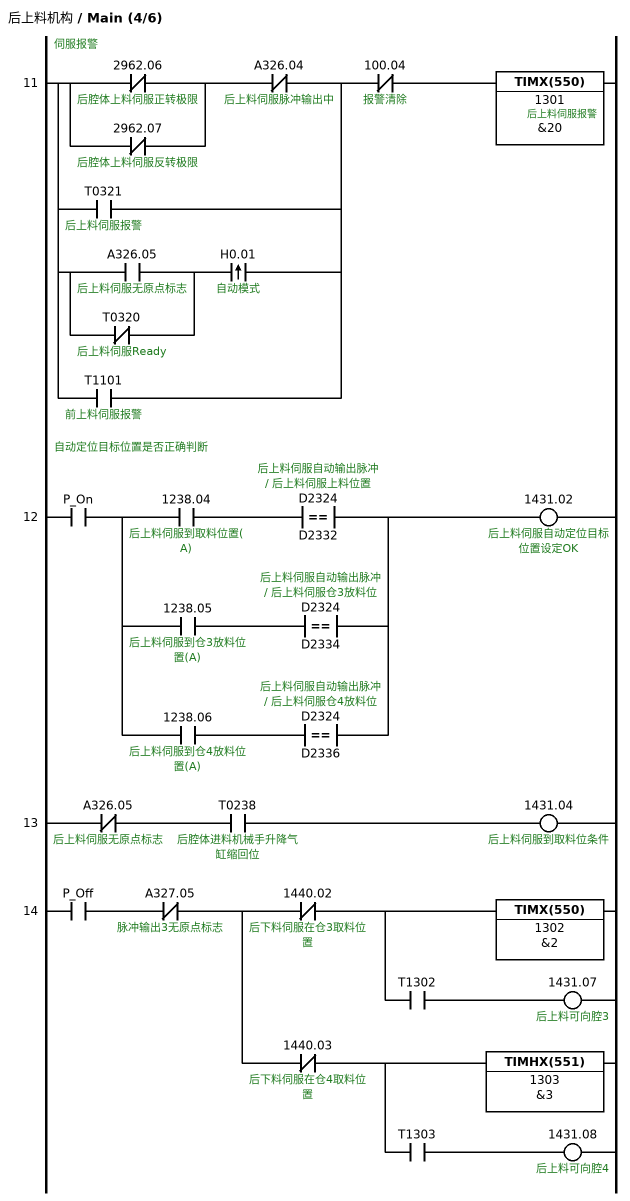
; rung 11: 伺服报警
LDNOT 2962.06  ; 后腔体上料伺服正转极限
ORNOT 2962.07  ; 后腔体上料伺服反转极限
ANDNOT A326.04  ; 后上料伺服脉冲输出中
OR T0321  ; 后上料伺服报警
LD A326.05  ; 后上料伺服无原点标志
ORNOT T0320  ; 后上料伺服Ready
@AND H0.01  ; 自动模式
ORLD
OR T1101  ; 前上料伺服报警
ANDNOT 100.04  ; 报警清除
TIMX(550) 1301 &20  ; 后上料伺服报警
; rung 12: 自动定位目标位置是否正确判断
LD P_On
LD 1238.04  ; 后上料伺服到取料位置(A)
AND=SL(303) D2324 D2332  ; 后上料伺服自动输出脉冲, 后上料伺服上料位置
LD 1238.05  ; 后上料伺服到仓3放料位置(A)
AND=SL(303) D2324 D2334  ; 后上料伺服自动输出脉冲, 后上料伺服仓3放料位
ORLD
LD 1238.06  ; 后上料伺服到仓4放料位置(A)
AND=SL(303) D2324 D2336  ; 后上料伺服自动输出脉冲, 后上料伺服仓4放料位
ORLD
ANDLD
OUT 1431.02  ; 后上料伺服自动定位目标位置设定OK
; rung 13
LDNOT A326.05  ; 后上料伺服无原点标志
AND T0238  ; 后腔体进料机械手升降气缸缩回位
OUT 1431.04  ; 后上料伺服到取料位条件
; rung 14
LD P_Off
ANDNOT A327.05  ; 脉冲输出3无原点标志
OUT TR0
ANDNOT 1440.02  ; 后下料伺服在仓3取料位置
TIMX(550) 1302 &2
AND T1302
OUT 1431.07  ; 后上料可向腔3
LD TR0
ANDNOT 1440.03  ; 后下料伺服在仓4取料位置
TIMHX(551) 1303 &3
AND T1303
OUT 1431.08  ; 后上料可向腔4

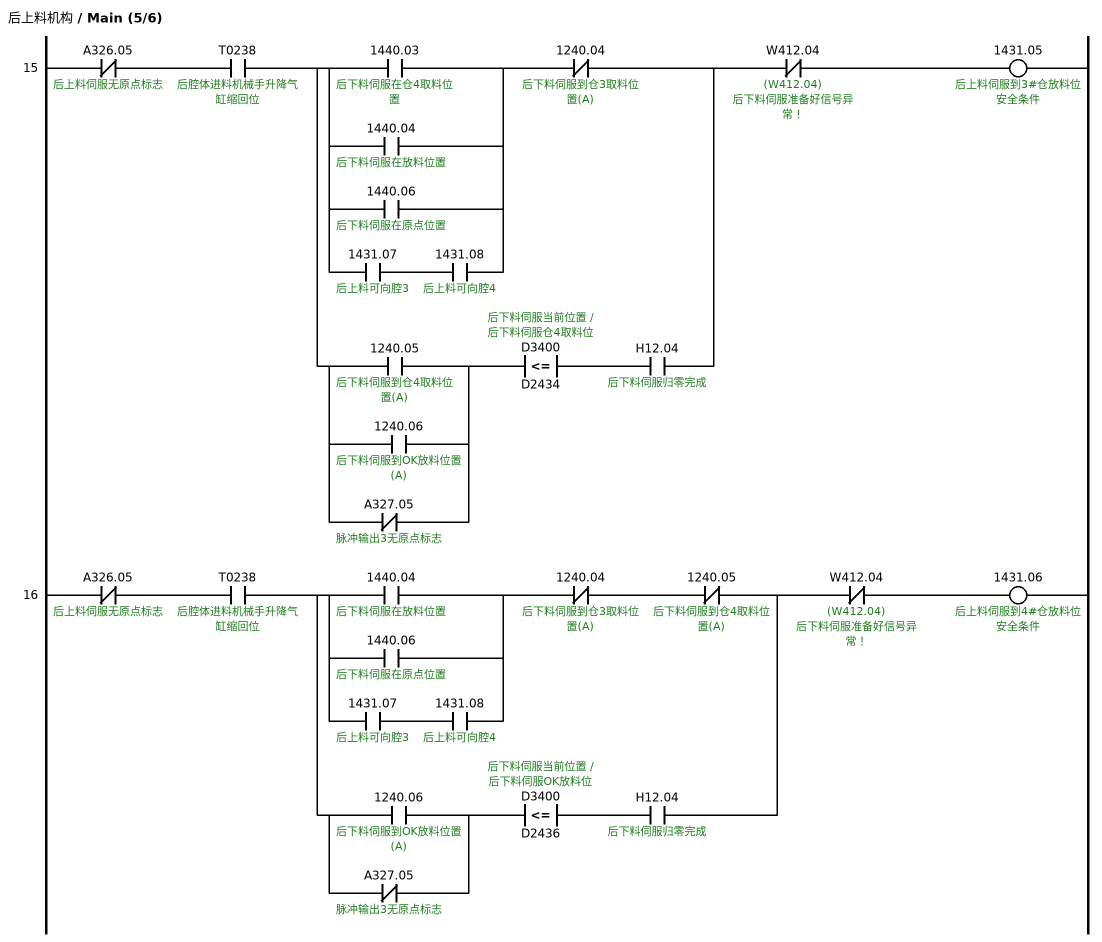
; rung 15
LDNOT A326.05  ; 后上料伺服无原点标志
AND T0238  ; 后腔体进料机械手升降气缸缩回位
LD 1440.03  ; 后下料伺服在仓4取料位置
OR 1440.04  ; 后下料伺服在放料位置
OR 1440.06  ; 后下料伺服在原点位置
LD 1431.07  ; 后上料可向腔3
AND 1431.08  ; 后上料可向腔4
ORLD
ANDNOT 1240.04  ; 后下料伺服到仓3取料位置(A)
LD 1240.05  ; 后下料伺服到仓4取料位置(A)
OR 1240.06  ; 后下料伺服到OK放料位置(A)
ORNOT A327.05  ; 脉冲输出3无原点标志
AND<=SL(318) D3400 D2434  ; 后下料伺服当前位置, 后下料伺服仓4取料位
AND H12.04  ; 后下料伺服归零完成
ORLD
ANDLD
ANDNOT W412.04  ; (W412.04) 后下料伺服准备好信号异常！
OUT 1431.05  ; 后上料伺服到3#仓放料位安全条件
; rung 16
LDNOT A326.05  ; 后上料伺服无原点标志
AND T0238  ; 后腔体进料机械手升降气缸缩回位
LD 1440.04  ; 后下料伺服在放料位置
OR 1440.06  ; 后下料伺服在原点位置
LD 1431.07  ; 后上料可向腔3
AND 1431.08  ; 后上料可向腔4
ORLD
ANDNOT 1240.04  ; 后下料伺服到仓3取料位置(A)
ANDNOT 1240.05  ; 后下料伺服到仓4取料位置(A)
LD 1240.06  ; 后下料伺服到OK放料位置(A)
ORNOT A327.05  ; 脉冲输出3无原点标志
AND<=SL(318) D3400 D2436  ; 后下料伺服当前位置, 后下料伺服OK放料位
AND H12.04  ; 后下料伺服归零完成
ORLD
ANDLD
ANDNOT W412.04  ; (W412.04) 后下料伺服准备好信号异常！
OUT 1431.06  ; 后上料伺服到4#仓放料位安全条件

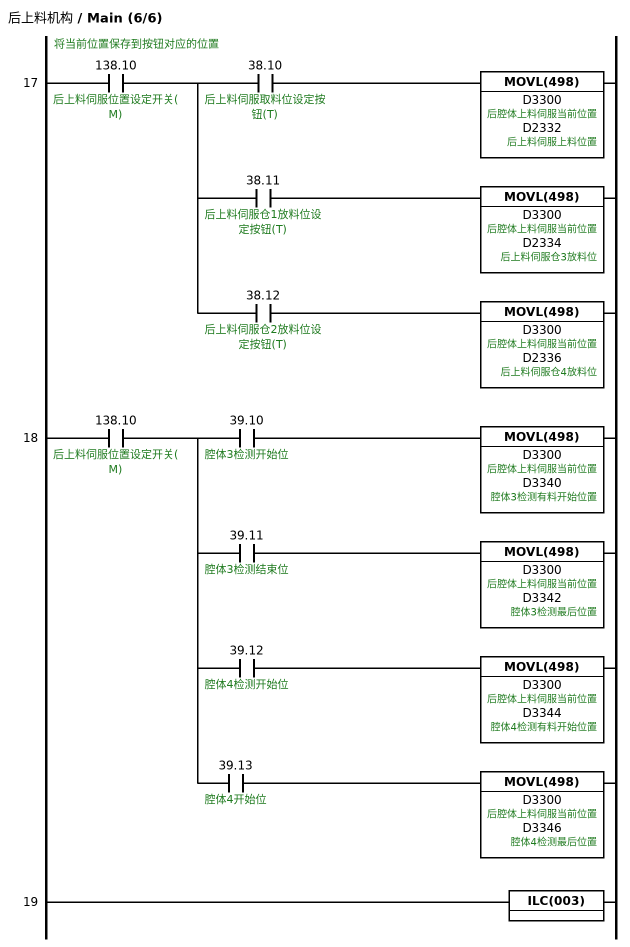
; rung 17: 将当前位置保存到按钮对应的位置
LD 138.10  ; 后上料伺服位置设定开关(M)
OUT TR0
AND 38.10  ; 后上料伺服取料位设定按钮(T)
MOVL(498) D3300 D2332  ; 后腔体上料伺服当前位置, 后上料伺服上料位置
LD TR0
AND 38.11  ; 后上料伺服仓1放料位设定按钮(T)
MOVL(498) D3300 D2334  ; 后腔体上料伺服当前位置, 后上料伺服仓3放料位
LD TR0
AND 38.12  ; 后上料伺服仓2放料位设定按钮(T)
MOVL(498) D3300 D2336  ; 后腔体上料伺服当前位置, 后上料伺服仓4放料位
; rung 18
LD 138.10  ; 后上料伺服位置设定开关(M)
OUT TR0
AND 39.10  ; 腔体3检测开始位
MOVL(498) D3300 D3340  ; 后腔体上料伺服当前位置, 腔体3检测有料开始位置
LD TR0
AND 39.11  ; 腔体3检测结束位
MOVL(498) D3300 D3342  ; 后腔体上料伺服当前位置, 腔体3检测最后位置
LD TR0
AND 39.12  ; 腔体4检测开始位
MOVL(498) D3300 D3344  ; 后腔体上料伺服当前位置, 腔体4检测有料开始位置
LD TR0
AND 39.13  ; 腔体4开始位
MOVL(498) D3300 D3346  ; 后腔体上料伺服当前位置, 腔体4检测最后位置
; rung 19
ILC(003)

### Section 工站复位

